TYPE ST_WaferTransferCtrl :
STRUCT
	Ctrl : ST_ServiceCtrl;
	Param : ST_WaferTransferParam;
	Signal : ST_TransferHandshakeSignal;
END_STRUCT
END_TYPE

(* stored: Version 1.1.0.1, ProductVersion 3.1.4026.18
   DUT ST_WaferTransferCtrl: Id {fbebe599-2e1e-42f5-9f7c-1dc0ab4296c0} *)
